// TIA Portal V20 export
// export: Created 2025-12-01T14:57:30.7717214Z, ExportSetting None, DisplayName Totally Integrated Automation Portal, DisplayVersion V20 Update 3, DisplayName TIA Portal Openness, DisplayVersion V20 Update 3, DisplayName TIA Portal Version Control Interface, DisplayVersion V20 Update 3, DisplayName STEP 7 Professional, DisplayVersion V20 Update 3, DisplayName STEP 7 Safety, DisplayVersion V20 Update 2, DisplayName WinCC Basic/Comfort/Advanced, DisplayVersion V20 Update 3, DisplayName WinCC Professional, DisplayVersion V20 Update 3, DisplayName WinCC Unified, DisplayVersion V20 Update 3
DATA_BLOCK "DB1700_Mesas_Fuentes"   // DB1700
{ S7_Optimized_Access := 'FALSE' }
// stored: AutoNumber false
   VAR
      Num_de_posicion_en_la_linea : Byte;   // Las tarjetas dentro de las lineas que tengan este numero, podran moverse
      Mesa { ExternalAccessible := 'False'; ExternalVisible := 'False'; ExternalWritable := 'False'} : Array[1..500] of "Fuentes_Lineas";
   END_VAR
BEGIN
   Mesa[1..7].Fuente := '2020';
   Mesa[8..25].Fuente := '2017';
   Mesa[26..33].Fuente := '2020';
   Mesa[34..35].Fuente := '2046';
   Mesa[37..45].Fuente := '2046';
   Mesa[50].Fuente := '2044';
   Mesa[51..65].Fuente := '3004';
   Mesa[66..71].Fuente := '3006';
   Mesa[73..82].Fuente := '3006';
   Mesa[90..95].Fuente := '7019';
   Mesa[96..105].Fuente := '7003';
   Mesa[106..119].Fuente := '7016';
   Mesa[120..125].Fuente := '7019';
   Mesa[300..305].Fuente := '2008A';
   Mesa[310..315].Fuente := '2008B';
   Mesa[320..325].Fuente := '2008C';
   Mesa[330..335].Fuente := '2008D';
   Mesa[400..405].Fuente := '7005A';
   Mesa[410..415].Fuente := '7005B';
   Mesa[420..425].Fuente := '7005C';
   Mesa[430..435].Fuente := '7005D';
   Mesa[1..3].Linea := 2;
   Mesa[4..7].Linea := 1;
   Mesa[8..12].Linea := 3;
   Mesa[13..16].Linea := 4;
   Mesa[17..20].Linea := 2;
   Mesa[21..25].Linea := 1;
   Mesa[26..30].Linea := 3;
   Mesa[31..33].Linea := 4;
   Mesa[34..35].Linea := 1;
   Mesa[37..38].Linea := 1;
   Mesa[39].Linea := 2;
   Mesa[40..42].Linea := 3;
   Mesa[43..45].Linea := 4;
   Mesa[50..54].Linea := 1;
   Mesa[55..58].Linea := 2;
   Mesa[59..62].Linea := 3;
   Mesa[63..65].Linea := 4;
   Mesa[66..69].Linea := 1;
   Mesa[70..71].Linea := 2;
   Mesa[73].Linea := 3;
   Mesa[74..76].Linea := 2;
   Mesa[77..80].Linea := 4;
   Mesa[81..82].Linea := 3;
   Mesa[90..93].Linea := 3;
   Mesa[94..95].Linea := 2;
   Mesa[96..99].Linea := 1;
   Mesa[100..102].Linea := 2;
   Mesa[103..105].Linea := 3;
   Mesa[106..108].Linea := 1;
   Mesa[109..111].Linea := 2;
   Mesa[112..115].Linea := 3;
   Mesa[116..119].Linea := 4;
   Mesa[120..123].Linea := 1;
   Mesa[124..125].Linea := 2;
   Mesa[300].Linea := 2;
   Mesa[301].Linea := 3;
   Mesa[302..305].Linea := 1;
   Mesa[310].Linea := 2;
   Mesa[311].Linea := 3;
   Mesa[312..315].Linea := 1;
   Mesa[320].Linea := 2;
   Mesa[321].Linea := 3;
   Mesa[322..325].Linea := 1;
   Mesa[330].Linea := 2;
   Mesa[331].Linea := 3;
   Mesa[332..335].Linea := 1;
   Mesa[400..403].Linea := 1;
   Mesa[404].Linea := 2;
   Mesa[405].Linea := 3;
   Mesa[410..413].Linea := 1;
   Mesa[414].Linea := 2;
   Mesa[415].Linea := 3;
   Mesa[420..423].Linea := 1;
   Mesa[424].Linea := 2;
   Mesa[425].Linea := 3;
   Mesa[430..433].Linea := 1;
   Mesa[434].Linea := 2;
   Mesa[435].Linea := 3;
   Mesa[1].Posicion := 3;
   Mesa[2].Posicion := 2;
   Mesa[3].Posicion := 1;
   Mesa[4].Posicion := 4;
   Mesa[5].Posicion := 3;
   Mesa[6].Posicion := 2;
   Mesa[7].Posicion := 1;
   Mesa[8].Posicion := 5;
   Mesa[9].Posicion := 4;
   Mesa[10].Posicion := 3;
   Mesa[11].Posicion := 2;
   Mesa[12..13].Posicion := 1;
   Mesa[14].Posicion := 2;
   Mesa[15].Posicion := 3;
   Mesa[16..17].Posicion := 4;
   Mesa[18].Posicion := 3;
   Mesa[19].Posicion := 2;
   Mesa[20..21].Posicion := 1;
   Mesa[22].Posicion := 2;
   Mesa[23].Posicion := 3;
   Mesa[24].Posicion := 4;
   Mesa[25].Posicion := 5;
   Mesa[26].Posicion := 1;
   Mesa[27].Posicion := 2;
   Mesa[28].Posicion := 3;
   Mesa[29].Posicion := 4;
   Mesa[30].Posicion := 5;
   Mesa[31].Posicion := 1;
   Mesa[32].Posicion := 3;
   Mesa[33].Posicion := 4;
   Mesa[34].Posicion := 1;
   Mesa[35].Posicion := 2;
   Mesa[37].Posicion := 1;
   Mesa[38].Posicion := 2;
   Mesa[39..40].Posicion := 1;
   Mesa[41].Posicion := 2;
   Mesa[42].Posicion := 3;
   Mesa[43].Posicion := 1;
   Mesa[44].Posicion := 2;
   Mesa[45].Posicion := 3;
   Mesa[50].Posicion := 1;
   Mesa[51].Posicion := 4;
   Mesa[52].Posicion := 3;
   Mesa[53].Posicion := 2;
   Mesa[54..56].Posicion := 1;
   Mesa[57].Posicion := 3;
   Mesa[58].Posicion := 4;
   Mesa[59].Posicion := 1;
   Mesa[60].Posicion := 2;
   Mesa[61].Posicion := 3;
   Mesa[62].Posicion := 4;
   Mesa[63].Posicion := 1;
   Mesa[64].Posicion := 2;
   Mesa[65].Posicion := 3;
   Mesa[66].Posicion := 4;
   Mesa[67].Posicion := 3;
   Mesa[68].Posicion := 2;
   Mesa[69].Posicion := 1;
   Mesa[70].Posicion := 2;
   Mesa[71].Posicion := 1;
   Mesa[73].Posicion := 1;
   Mesa[74].Posicion := 3;
   Mesa[75].Posicion := 4;
   Mesa[76..77].Posicion := 5;
   Mesa[78].Posicion := 4;
   Mesa[79].Posicion := 3;
   Mesa[80..81].Posicion := 2;
   Mesa[82].Posicion := 3;
   Mesa[83].Posicion := 1;
   Mesa[84].Posicion := 2;
   Mesa[90].Posicion := 4;
   Mesa[91].Posicion := 3;
   Mesa[92].Posicion := 2;
   Mesa[93].Posicion := 1;
   Mesa[94].Posicion := 4;
   Mesa[95].Posicion := 3;
   Mesa[96].Posicion := 4;
   Mesa[97].Posicion := 3;
   Mesa[98].Posicion := 2;
   Mesa[99..100].Posicion := 1;
   Mesa[101].Posicion := 2;
   Mesa[102].Posicion := 3;
   Mesa[103].Posicion := 1;
   Mesa[104].Posicion := 2;
   Mesa[105].Posicion := 3;
   Mesa[106].Posicion := 1;
   Mesa[107].Posicion := 2;
   Mesa[108].Posicion := 3;
   Mesa[109].Posicion := 1;
   Mesa[110].Posicion := 2;
   Mesa[111].Posicion := 3;
   Mesa[112].Posicion := 4;
   Mesa[113].Posicion := 3;
   Mesa[114].Posicion := 2;
   Mesa[115..116].Posicion := 1;
   Mesa[117].Posicion := 2;
   Mesa[118].Posicion := 3;
   Mesa[119..120].Posicion := 4;
   Mesa[121].Posicion := 3;
   Mesa[122].Posicion := 2;
   Mesa[123..124].Posicion := 1;
   Mesa[125].Posicion := 2;
   Mesa[300..302].Posicion := 1;
   Mesa[303].Posicion := 2;
   Mesa[304].Posicion := 3;
   Mesa[305].Posicion := 4;
   Mesa[310..312].Posicion := 1;
   Mesa[313].Posicion := 2;
   Mesa[314].Posicion := 3;
   Mesa[315].Posicion := 4;
   Mesa[320..322].Posicion := 1;
   Mesa[323].Posicion := 2;
   Mesa[324].Posicion := 3;
   Mesa[325].Posicion := 4;
   Mesa[330..332].Posicion := 1;
   Mesa[333].Posicion := 2;
   Mesa[334].Posicion := 3;
   Mesa[335].Posicion := 4;
   Mesa[400].Posicion := 1;
   Mesa[401].Posicion := 2;
   Mesa[402].Posicion := 3;
   Mesa[403].Posicion := 4;
   Mesa[404..405].Posicion := 1;
   Mesa[410].Posicion := 1;
   Mesa[411].Posicion := 2;
   Mesa[412].Posicion := 3;
   Mesa[413].Posicion := 4;
   Mesa[414..415].Posicion := 1;
   Mesa[420].Posicion := 1;
   Mesa[421].Posicion := 2;
   Mesa[422].Posicion := 3;
   Mesa[423].Posicion := 4;
   Mesa[424..425].Posicion := 1;
   Mesa[430].Posicion := 1;
   Mesa[431].Posicion := 2;
   Mesa[432].Posicion := 3;
   Mesa[433].Posicion := 4;
   Mesa[434..435].Posicion := 1;
END_DATA_BLOCK
